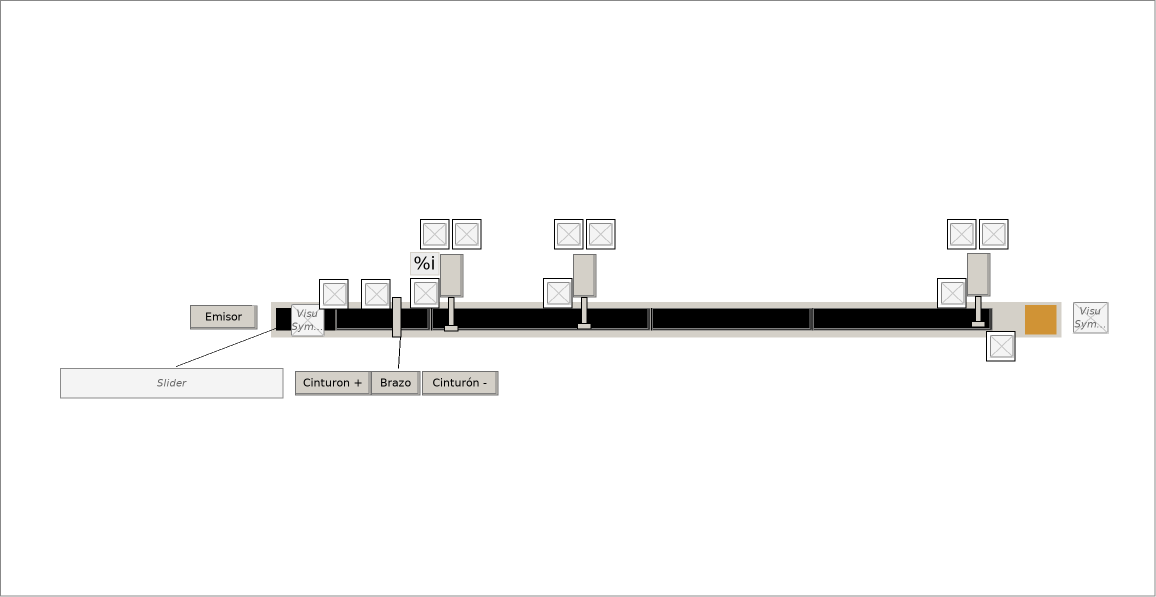
VISUALIZATION Entrada_Manual  // 1156x597
    Button (190,305 67x24), "Emisor", colour toggle: GVL.Emitter_1, pressed state: GVL.Emitter_1
        OnMouseClick: toggle GVL.Emitter_1
    Rectangle (252,287 92x18)
    Slider (60,368 223x30), variable: GVL.Belt_Conveyor_2m_1, scale -10..10
    Button (371,371 49x24), "Brazo", colour toggle: GVL.Pivot_Arm_Sorter_1_Turn, pressed state: GVL.Pivot_Arm_Sorter_1_Turn
        OnMouseClick: toggle GVL.Pivot_Arm_Sorter_1_Turn
    Button (295,371 76x24), "Cinturon +", colour toggle: GVL.Pivot_Arm_Sorter_1_Belt_mas, pressed state: GVL.Pivot_Arm_Sorter_1_Belt_mas
        OnMouseClick: toggle GVL.Pivot_Arm_Sorter_1_Belt_mas
    Button (422,371 76x24), "Cinturón -", colour toggle: GVL.Pivot_Arm_Sorter_1_Belt_menos, pressed state: GVL.Pivot_Arm_Sorter_1_Belt_menos
        OnMouseClick: toggle GVL.Pivot_Arm_Sorter_1_Belt_menos
    Line (401,320) (398,368)
    InvisibleInput (369,461 77x136)
    InvisibleInput (1141,334 15x136)
    InvisibleInput (1064,298 50x41)
    Rectangle (1033,330 35x70), angle 90
    Rectangle (271,302 724x35)
    RoundedRectangle (810,308 179x22), colour toggle: GVL.Belt_Conveyor_6m_5
    RoundedRectangle (276,308 59x22), colour toggle: GVL.Emitter_1
        OnMouseClick: toggle GVL.Emitter_1
    Image (291,304 33x32), image: VisuSymbols.Symbols.ForwardStandard
    Image (1073,302 35x31), image: VisuSymbols.Symbols.ArrowCircle2RightUpDown
    RoundedRectangle (1025,305 31x29)
    RoundedRectangle (431,308 219x22), colour toggle: GVL.Belt_Conveyor_6m_1
    RoundedRectangle (651,308 160x22), colour toggle: GVL.Belt_Conveyor_6m_4
    Rectangle (440,254 23x43)
    Rectangle (573,254 23x43)
    Rectangle (967,253 23x43)
    Button (336,308 94x22), colour toggle: GVL.Belt_Conveyor_4m_1, pressed state: GVL.Belt_Conveyor_4m_1
        OnMouseClick: toggle GVL.Belt_Conveyor_4m_1
    Rectangle (377,313 40x9), angle 90, colour toggle: GVL.Belt_Conveyor_4m_1
    Line (176,366) (286,324)
    Button (440,254 23x43), colour toggle: GVL.Pusher_1, pressed state: GVL.Pusher_1
        OnMouseClick: toggle GVL.Pusher_1
    Button (573,254 23x43), colour toggle: GVL.Pusher_2, pressed state: GVL.Pusher_2
        OnMouseClick: toggle GVL.Pusher_2
    Button (967,253 23x43), colour toggle: GVL.Pusher_3, pressed state: GVL.Pusher_3
        OnMouseClick: toggle GVL.Pusher_3
    Button (432,308 218x22), colour toggle: GVL.Belt_Conveyor_6m_1, pressed state: GVL.Belt_Conveyor_6m_1
        OnMouseClick: toggle GVL.Belt_Conveyor_6m_1
    Rectangle (448,297 6x29)
    Rectangle (581,297 6x29)
    Button (652,308 160x22), colour toggle: GVL.Belt_Conveyor_6m_4, pressed state: GVL.Belt_Conveyor_6m_4
        OnMouseClick: toggle GVL.Belt_Conveyor_6m_4
    Button (813,308 179x22), colour toggle: GVL.Belt_Conveyor_6m_5, pressed state: GVL.Belt_Conveyor_6m_5
        OnMouseClick: toggle GVL.Belt_Conveyor_6m_5
    Rectangle (975,296 6x29)
    Rectangle (985,323 6x14), angle 270
    Group (319,279 29x30)
        RoundedRectangle (0,0 29x30), colour toggle: GVL.Diffuse_Sensor_0
        Image (4,4 23x22), image: VisuSymbols.Symbols.RSS1
    Group (361,279 29x30)
        RoundedRectangle (0,0 29x30), colour toggle: GVL.Diffuse_Sensor_1
        Image (4,4 23x22), image: VisuSymbols.Symbols.RSS1
    Group (410,278 29x30)
        RoundedRectangle (0,0 29x30), colour toggle: GVL.Diffuse_Sensor_2
        Image (4,4 23x22), image: VisuSymbols.Symbols.RSS1
    Group (543,278 29x30)
        RoundedRectangle (0,0 29x30), colour toggle: GVL.Diffuse_Sensor_3
        Image (4,4 23x22), image: VisuSymbols.Symbols.RSS1
    Group (937,278 29x30)
        RoundedRectangle (0,0 29x30), colour toggle: GVL.Diffuse_Sensor_4
        Image (4,4 23x22), image: VisuSymbols.Symbols.RSS1
    Group (986,331 29x30)
        RoundedRectangle (0,0 29x30), colour toggle: GVL.Diffuse_Sensor_8
        Image (4,4 23x22), image: VisuSymbols.Symbols.RSS1
    Group (452,219 29x30)
        RoundedRectangle (0,0 29x30), colour toggle: GVL.Pusher_1_Front_Limit
        Image (3,4 23x22), image: VisuSymbols.Symbols.ArrowBoldDown
    Group (420,219 29x30)
        RoundedRectangle (0,0 29x30), colour toggle: GVL.Pusher_1_Back_Limit
        Image (3,4 23x22), image: VisuSymbols.Symbols.ArrowBoldUp
    Group (586,219 29x30)
        RoundedRectangle (0,0 29x30), colour toggle: GVL.Pusher_2_Front_Limit
        Image (3,4 23x22), image: VisuSymbols.Symbols.ArrowBoldDown
    Group (554,219 29x30)
        RoundedRectangle (0,0 29x30), colour toggle: GVL.Pusher_2_Back_Limit
        Image (3,4 23x22), image: VisuSymbols.Symbols.ArrowBoldUp
    Group (979,219 29x30)
        RoundedRectangle (0,0 29x30), colour toggle: GVL.Pusher_3_Front_Limit
        Image (3,4 23x22), image: VisuSymbols.Symbols.ArrowBoldDown
    Group (947,219 29x30)
        RoundedRectangle (0,0 29x30), colour toggle: GVL.Pusher_3_Back_Limit
        Image (3,4 23x22), image: VisuSymbols.Symbols.ArrowBoldUp
    Rectangle (410,252 29x23), "%i", text variable: GVL.Vision_Sensor_1
        p4168582468: GVL.Vision_Sensor_1
    Rectangle (455,324 6x14), angle 270
    Rectangle (590,324 6x14), angle 270
END_VISUALIZATION

(* stored: Version 1.1.0.1, ProductVersion 3.1.4024.12
   Visu Entrada_Manual: Id {a6ba39d0-95df-4eda-b151-0b10a44f364d} *)
